FUNCTION_BLOCK FB_HVFAStorage
VAR_INPUT
END_VAR
VAR_OUTPUT
END_VAR
VAR
	UpperTemperatureSensor : FB_TemperatureSensor;
	LowerTemperatureSensor : FB_TemperatureSensor;
END_VAR

//get sensor inputs
UpperTemperatureSensor.SetState_AI();
LowerTemperatureSensor.SetState_AI();

END_FUNCTION_BLOCK

(* stored: Version 1.1.0.1, ProductVersion 3.1.4024.9
   POU FB_HVFAStorage: Id {4e82d7a1-f7f2-424a-a2d3-5178f16a7cfd}, SpecialFunc None *)
